// TIA Portal V19 export
VAR_GLOBAL   // PLC tag table "Safety"
END_VAR
